// Mitsubishi GX Works2 project: 检测肥料有无   PLC: FX3U/FX3UC

PROGRAM MAIN
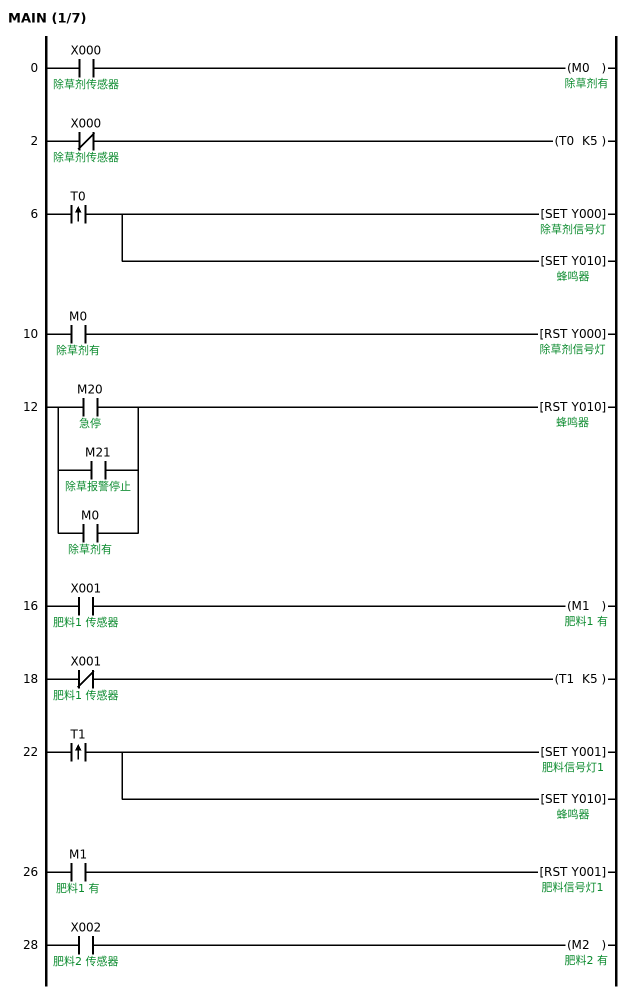
0     LD      X000  ; 除草剂传感器
      OUT     M0  ; 除草剂有
2     LDI     X000  ; 除草剂传感器
      OUT     T0 K5
6     LDP     T0
      SET     Y000  ; 除草剂信号灯
      SET     Y010  ; 蜂鸣器
10    LD      M0  ; 除草剂有
      RST     Y000  ; 除草剂信号灯
12    LD      M20  ; 急停
      OR      M21  ; 除草报警停止
      OR      M0  ; 除草剂有
      RST     Y010  ; 蜂鸣器
16    LD      X001  ; 肥料1 传感器
      OUT     M1  ; 肥料1 有
18    LDI     X001  ; 肥料1 传感器
      OUT     T1 K5
22    LDP     T1
      SET     Y001  ; 肥料信号灯1
      SET     Y010  ; 蜂鸣器
26    LD      M1  ; 肥料1 有
      RST     Y001  ; 肥料信号灯1
28    LD      X002  ; 肥料2 传感器
      OUT     M2  ; 肥料2 有
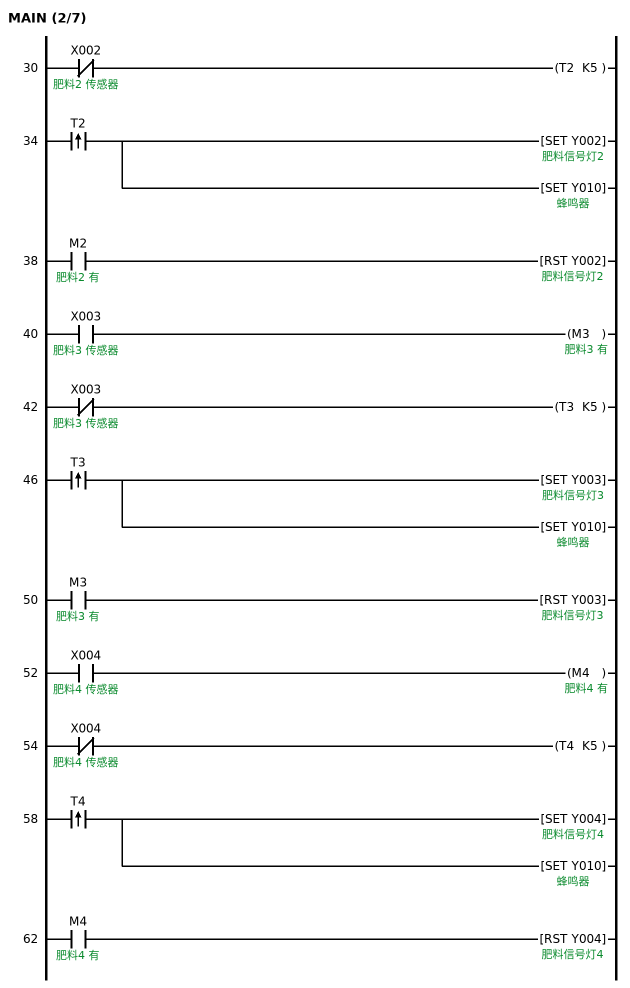
30    LDI     X002  ; 肥料2 传感器
      OUT     T2 K5
34    LDP     T2
      SET     Y002  ; 肥料信号灯2
      SET     Y010  ; 蜂鸣器
38    LD      M2  ; 肥料2 有
      RST     Y002  ; 肥料信号灯2
40    LD      X003  ; 肥料3 传感器
      OUT     M3  ; 肥料3 有
42    LDI     X003  ; 肥料3 传感器
      OUT     T3 K5
46    LDP     T3
      SET     Y003  ; 肥料信号灯3
      SET     Y010  ; 蜂鸣器
50    LD      M3  ; 肥料3 有
      RST     Y003  ; 肥料信号灯3
52    LD      X004  ; 肥料4 传感器
      OUT     M4  ; 肥料4 有
54    LDI     X004  ; 肥料4 传感器
      OUT     T4 K5
58    LDP     T4
      SET     Y004  ; 肥料信号灯4
      SET     Y010  ; 蜂鸣器
62    LD      M4  ; 肥料4 有
      RST     Y004  ; 肥料信号灯4
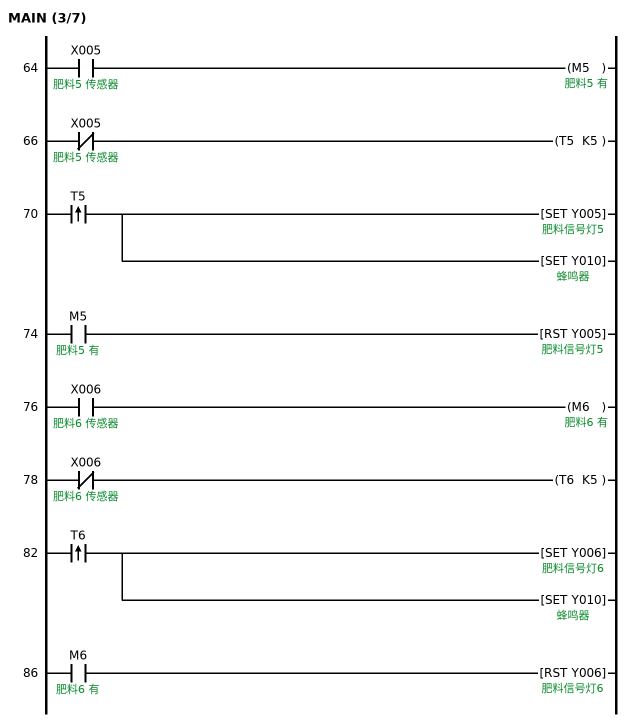
64    LD      X005  ; 肥料5 传感器
      OUT     M5  ; 肥料5 有
66    LDI     X005  ; 肥料5 传感器
      OUT     T5 K5
70    LDP     T5
      SET     Y005  ; 肥料信号灯5
      SET     Y010  ; 蜂鸣器
74    LD      M5  ; 肥料5 有
      RST     Y005  ; 肥料信号灯5
76    LD      X006  ; 肥料6 传感器
      OUT     M6  ; 肥料6 有
78    LDI     X006  ; 肥料6 传感器
      OUT     T6 K5
82    LDP     T6
      SET     Y006  ; 肥料信号灯6
      SET     Y010  ; 蜂鸣器
86    LD      M6  ; 肥料6 有
      RST     Y006  ; 肥料信号灯6
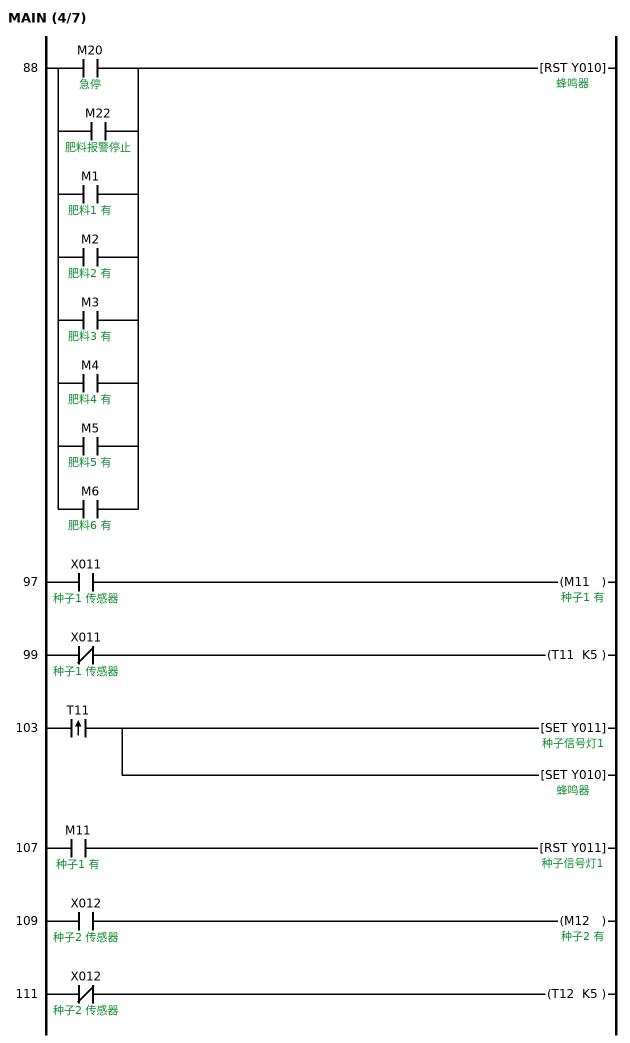
88    LD      M20  ; 急停
      OR      M22  ; 肥料报警停止
      OR      M1  ; 肥料1 有
      OR      M2  ; 肥料2 有
      OR      M3  ; 肥料3 有
      OR      M4  ; 肥料4 有
      OR      M5  ; 肥料5 有
      OR      M6  ; 肥料6 有
      RST     Y010  ; 蜂鸣器
97    LD      X011  ; 种子1 传感器
      OUT     M11  ; 种子1 有
99    LDI     X011  ; 种子1 传感器
      OUT     T11 K5
103   LDP     T11
      SET     Y011  ; 种子信号灯1
      SET     Y010  ; 蜂鸣器
107   LD      M11  ; 种子1 有
      RST     Y011  ; 种子信号灯1
109   LD      X012  ; 种子2 传感器
      OUT     M12  ; 种子2 有
111   LDI     X012  ; 种子2 传感器
      OUT     T12 K5
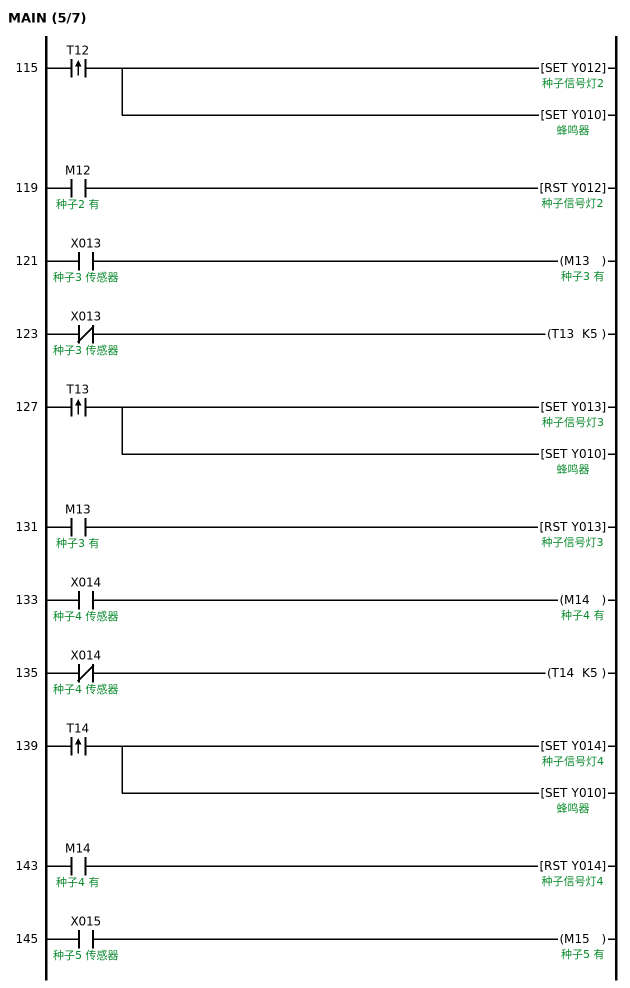
115   LDP     T12
      SET     Y012  ; 种子信号灯2
      SET     Y010  ; 蜂鸣器
119   LD      M12  ; 种子2 有
      RST     Y012  ; 种子信号灯2
121   LD      X013  ; 种子3 传感器
      OUT     M13  ; 种子3 有
123   LDI     X013  ; 种子3 传感器
      OUT     T13 K5
127   LDP     T13
      SET     Y013  ; 种子信号灯3
      SET     Y010  ; 蜂鸣器
131   LD      M13  ; 种子3 有
      RST     Y013  ; 种子信号灯3
133   LD      X014  ; 种子4 传感器
      OUT     M14  ; 种子4 有
135   LDI     X014  ; 种子4 传感器
      OUT     T14 K5
139   LDP     T14
      SET     Y014  ; 种子信号灯4
      SET     Y010  ; 蜂鸣器
143   LD      M14  ; 种子4 有
      RST     Y014  ; 种子信号灯4
145   LD      X015  ; 种子5 传感器
      OUT     M15  ; 种子5 有
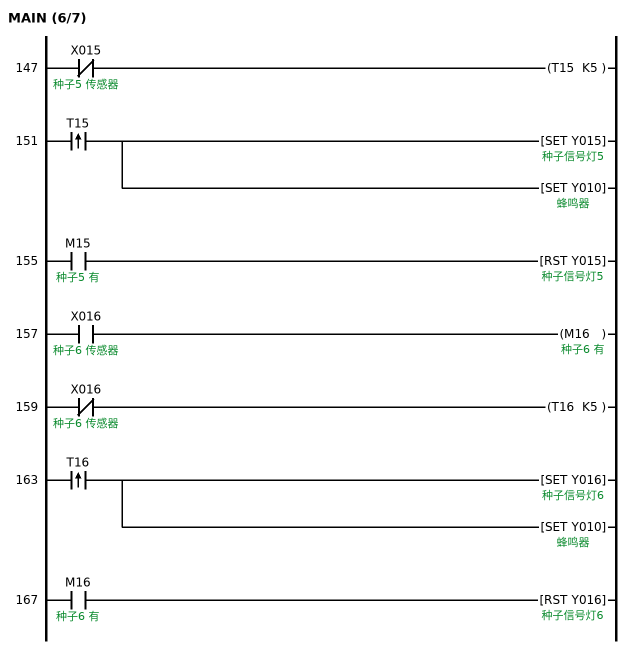
147   LDI     X015  ; 种子5 传感器
      OUT     T15 K5
151   LDP     T15
      SET     Y015  ; 种子信号灯5
      SET     Y010  ; 蜂鸣器
155   LD      M15  ; 种子5 有
      RST     Y015  ; 种子信号灯5
157   LD      X016  ; 种子6 传感器
      OUT     M16  ; 种子6 有
159   LDI     X016  ; 种子6 传感器
      OUT     T16 K5
163   LDP     T16
      SET     Y016  ; 种子信号灯6
      SET     Y010  ; 蜂鸣器
167   LD      M16  ; 种子6 有
      RST     Y016  ; 种子信号灯6
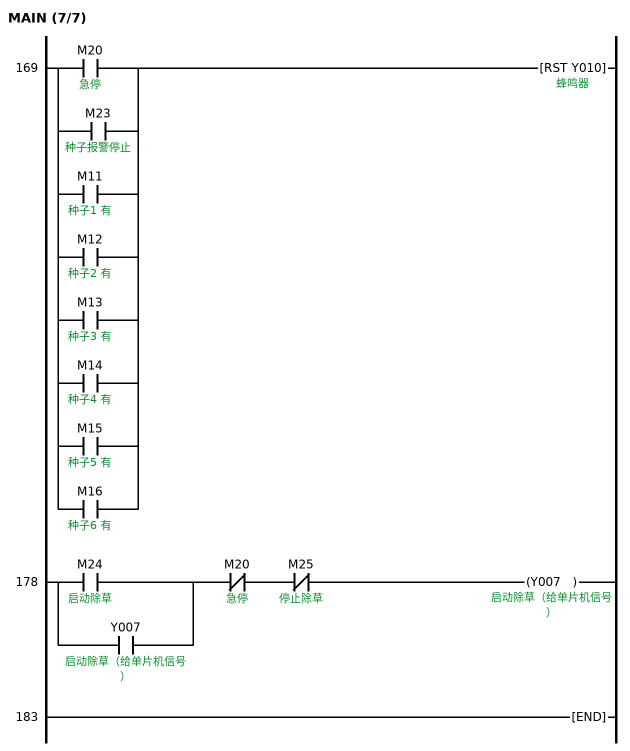
169   LD      M20  ; 急停
      OR      M23  ; 种子报警停止
      OR      M11  ; 种子1 有
      OR      M12  ; 种子2 有
      OR      M13  ; 种子3 有
      OR      M14  ; 种子4 有
      OR      M15  ; 种子5 有
      OR      M16  ; 种子6 有
      RST     Y010  ; 蜂鸣器
178   LD      M24  ; 启动除草
      OR      Y007  ; 启动除草（给单片机信号）
      ANI     M20  ; 急停
      ANI     M25  ; 停止除草
      OUT     Y007  ; 启动除草（给单片机信号）
183   END
END_PROGRAM

// device comments not shown above
M7  ; 肥料7 有
